{attribute 'qualified_only'}
VAR_GLOBAL
	// Meldeleuchte "Störung"
	P1: BOOL;
	// Motor Linkslauf
	Q1: BOOL;
	// Motor Rechtslauf
	Q2: BOOL;
END_VAR

(* stored: Version 1.1.0.1, ProductVersion 3.1.4022.7
   GVL AdsOutput: Id {efa3d63a-96e1-4204-b1e7-9f3703bd4f03} *)
